{attribute 'enable_dynamic_creation'}
FUNCTION_BLOCK FB_Stamp EXTENDS FB_PieceBase
VAR_INPUT
END_VAR
VAR_OUTPUT
END_VAR
VAR
END_VAR

METHOD FB_init : BOOL
VAR_INPUT
	bInitRetains : BOOL; // if TRUE, the retain variables are initialized (warm start / cold start)
	bInCopyCode : BOOL;  // if TRUE, the instance afterwards gets moved into the copy code (online change)
END_VAR
eObjectType := E_ObjectType.OBJECTTYPE_Stamp;
eObjectGroup := E_ObjectGroup.OBJECTGROUP_Piece;
END_METHOD

END_FUNCTION_BLOCK

(* stored: Version 1.1.0.1, ProductVersion 3.1.4022.18
   POU FB_Stamp: Id {681cb9ab-6215-487e-8c52-073187215eaf}, SpecialFunc None
   Method FB_init: Id {17d73328-dd20-4ffa-a1f1-a2851255ad38} *)
